(* PLC project Controller, Beckhoff Automation GmbH TwinCAT PLC Control 3.5.10.30 *)
(* stored: creationDateTime 2019-09-13T11:24:53.5838063, modificationDateTime 2019-09-13T11:24:53.588806 *)

TYPE ST_TcXboxController :
STRUCT
	counter : UDINT;
	A : BOOL;
	B : BOOL;
	X : BOOL;
	Y : BOOL;
	LB : BOOL;
	RB : BOOL;
	BACK : BOOL;
	START : BOOL;
	DPAD_UP : BOOL;
	DPAD_DOWN : BOOL;
	DPAD_LEFT : BOOL;
	DPAD_RIGHT : BOOL;
	LEFT_THUMB : BOOL;
	RIGHT_THUMB : BOOL;
	LEFT_TRIGGER : REAL;
	RIGHT_TRIGGER : REAL;
	JOY_LX : REAL;
	JOY_LY : REAL;
	JOY_RX : REAL;
	JOY_RY : REAL;
END_STRUCT
END_TYPE
